TYPE ST_Camming :
	STRUCT
		camIn		   : MC_CamIn_V2;
		camOut		   : MC_CamOut;
		camPoints	   : ARRAY[1..94] OF MC_MotionFunctionPoint;
		camRef		   : MC_CAM_REF;
		camTableSelect : MC_CamTableSelect;
		camAdd		   : MC_CamAdd;
		camRemove	   : MC_CamRemove;
        camScaling     :  ST_CamScalingData;
	END_STRUCT
END_TYPE

(* stored: Version 1.1.0.1, ProductVersion 3.1.4026.21
   DUT ST_Camming: Id {9e594c57-3e05-48f9-ad7f-5ef832bb29a5} *)
